// TIA Portal V20 export
FUNCTION_BLOCK "FB_CommPLC_ISO"   // FB1100, SCL
{ S7_Optimized_Access := 'TRUE' }
// stored: AutoNumber false, MemoryReserve 100, SetENOAutomatically false
   VAR DB_SPECIFIC
      sSynchro_ULx { ExternalVisible := 'False'; ExternalWritable := 'False'} : Byte;   // Image of A_DBB[1000]
   END_VAR
   VAR
      sSynchro_ULx_WriteON { ExternalAccessible := 'False'; ExternalVisible := 'False'; ExternalWritable := 'False'} : Bool;
      sRT_FixtureVW_Rel : R_TRIG;
      sRT_FixtureVW_Req { S7_SetPoint := 'True'} : R_TRIG;
      sRT_GripperAvail { S7_SetPoint := 'True'} : R_TRIG;
      sAxisManagedByNC { S7_SetPoint := 'True'} : Bool;
      sAxisReservedbyNC : Bool;
   END_VAR
   VAR_TEMP
      tSynchro_ULx_ReadON : Bool;
      tReadError : Bool;
      tWriteError : Bool;
      tReadErrCode : Int;
      tWriteErrCode : Int;
   END_VAR
BEGIN

   REGION Read/Write Byte Cmd : $A_DBB[1000]
       // SYNCHRO_UL1
       // SYNCHRO_UL1 = 1 : Demande axes par NC (Mise à 1 par NC)
       // SYNCHRO_UL1 = 0 : Liberation axes par PLC (Mise à 0 par PLC)

       #sRT_GripperAvail(CLK := "DB_GestionGripper".sGripperStatus.Available);


       #sRT_FixtureVW_Req(CLK := (("DB_LoaderFixture".sFixtureMain.iGripperReadyForUnloading AND NOT "DB_WorkingModes".sFilling) // Gripper ready for Unloading
                          OR ("DB_LoaderFixture".sFixtureMain.iGripperReadyForLoading AND "DB_WorkingModes".sFilling)            // Gripper ready for Loading
                          OR #sRT_GripperAvail.Q                                                                                 // Gripper Available  
                          OR "DB_WorkingModes".sManu) AND #sSynchro_ULx.%X0);                                                    // Mode Manu
       IF #sRT_FixtureVW_Req.Q THEN
           #sSynchro_ULx.%X0 := FALSE;
           #sSynchro_ULx_WriteON := TRUE;
       END_IF;

       // SYNCHRO_UL2
       // SYNCHRO_UL2 = 1 : Liberation axes par NC (Mise à 1 par NC)
       // SYNCHRO_UL2 = 0 : Demande axes par PLC (Mise à 0 par PLC)   
       #sRT_FixtureVW_Rel(CLK := "DB_GestionGripper".sGripperStatus.Available AND #sSynchro_ULx.%X1); // Acquittement Liberation dès que Gripper Available
       IF #sRT_FixtureVW_Rel.Q THEN
           #sSynchro_ULx.%X1 := FALSE;
           #sSynchro_ULx_WriteON := TRUE;
       END_IF;

       // Axis reserved by NC
       IF #sRT_FixtureVW_Req.Q THEN
           #sAxisReservedbyNC := TRUE;
       ELSIF  #sRT_FixtureVW_Rel.Q OR "LBP_Chan1".A_Reset THEN
           #sAxisReservedbyNC := FALSE;
       END_IF;

       // Datas FOR Communication PLC <--> ISO
           // DEFINE xREAD_SYNCHRO_UL1         AS (($A_DBB[1000] B_AND 1)==1)
           // DEFINE xWRITE_ON_SYNCHRO_UL1     AS $A_DBB[1000]=$A_DBB[1000] B_OR 1
           // DEFINE xWRITE_OFF_SYNCHRO_UL1    AS $A_DBB[1000]=$A_DBB[1000] B_AND (255-1)

           // DEFINE xREAD_SYNCHRO_UL2         AS (($A_DBB[1000] B_AND 2)==2)
           // DEFINE xWRITE_ON_SYNCHRO_UL2     AS $A_DBB[1000]=$A_DBB[1000] B_OR 2
           // DEFINE xWRITE_OFF_SYNCHRO_UL2    AS $A_DBB[1000]=$A_DBB[1000] B_AND (255-2)
           // 


       // SYNCHRO_UL2 = 1 : Liberation axes par NC (Mise à 1 par NC)
       // SYNCHRO_UL2 = 0 : Demande axes par PLC (Mise à 0 par PLC)
       "LBP_TransferSelData"(Enable := #sSynchro_ULx_WriteON,
                             Funct := 4,
                             S7Var := #sSynchro_ULx,
                             IVAR1 := 1000,
                             IVAR2 := -1,
                             Error => #tWriteError,
                             ErrCode => #tWriteErrCode);

       IF NOT #sSynchro_ULx_WriteON THEN
           #tSynchro_ULx_ReadON := True;
       ELSE
           #tSynchro_ULx_ReadON := False;
       END_IF;
       IF (#sSynchro_ULx_WriteON AND NOT #tWriteError) THEN
           #sSynchro_ULx_WriteON := False;
       END_IF;

       "LBP_TransferSelData"(Enable := #tSynchro_ULx_ReadON,
                             Funct := 3,
                             S7Var := #sSynchro_ULx,
                             IVAR1 := 1000,
                             IVAR2 := -1,
                             Error => #tReadError,
                             ErrCode => #tReadErrCode);
   END_REGION
END_FUNCTION_BLOCK
